# EPICS autosave request: iocBoot/iocFX4/auto_settings.req
file "quadEM_IOC_settings.req",        P=$(P), R=$(R)
file "FX4_settings.req",               P=$(P), R=$(R)
